% RSLogix 500 project SW2014_AK.RSS, saved by version 12.00.00.00 %
PROJECT "PS8"    % processor: MicroLogix 1400 %

PROGRAM FILES
  LAD 2 "MAIN"  27 rungs  % Calls all system and subsystem routines %
  LAD 3 "CONSTANTS"  51 rungs  % Maintains the system constants %
  LAD 4 "DEFAULTS"  49 rungs  % Manages the system default values %
  LAD 5 "SYS_FAULTS"  43 rungs  % Monitors the system fault conditions %
  LAD 6 "SYSTEM"  50 rungs  % Controls the system %
  LAD 7 "PROCESSING"  33 rungs  % Runs the processing control %
  LAD 8 "MANUAL_CTL"  14 rungs  % Runs the manual valve control %
  LAD 10 "PURIFY"  36 rungs  % Operates the purify control %
  LAD 11 "REGEN"  79 rungs  % Operates the regen control %
  LAD 12 "REGEN_FLT"  47 rungs  % regen alarms and warnings %
  LAD 17 "BYPASS"  4 rungs  % Controls the bypass %
  LAD 18 "MIX PANEL"  9 rungs
  LAD 20 "ADS_A"  45 rungs  % Controls the Adsorber A %
  LAD 21 "ADS_A_FLT"  17 rungs  % Controls the Adsorber A faults %
  LAD 22 "ADS_B"  45 rungs  % Controld Adsorber B %
  LAD 23 "ADS_B_FLT"  17 rungs  % Controls the Adsorber B faults %
  LAD 24 "PREHEATER"  10 rungs
  LAD 25 "PH_FLT"  19 rungs
  LAD 26 "ADS_C"  45 rungs
  LAD 27 "ADS_C_FLT"  17 rungs
  LAD 28 "ADS_D"  45 rungs
  LAD 29 "ADS_D_FLT"  17 rungs
  LAD 49 "MODBUS"  38 rungs
  LAD 50 "PLC_FAULT"  2 rungs
  LAD 51 "REVERSE"  9 rungs

DATA FILES
  O0 OUTPUT  25 elements
  I1 INPUT  25 elements
  S2 STATUS  66 elements
  B3 BINARY  4 elements
  T4 TIMER  142 elements
  C5 COUNTER  22 elements
  R6 CONTROL  2 elements
  N7 SYSTEM CFG  140 elements  % Maintains the values that characterize the system %
  F8 FLOAT  3 elements
  N9 CONSTANTS  86 elements  % The collection of system and subsystem constants %
  N10 SYSTEM  30 elements  % Contain the values for system control %
  N11 PROCESS  10 elements  % Contains the values for the processing machine %
  N12 PURIFY  25 elements  % Contains the values required for purify %
  N13 REGEN  31 elements  % Contains the values required for regen %
  N14 BYPASS  2 elements
  N15 MANUAL CTL  6 elements  % Contains the data for the manual valve control %
  N16 ADSORBER_A  22 elements  % Contains the values for Adsorber A %
  N17 ADSORBER_B  22 elements  % Contains the values required for Adsorber B %
  N18 ADSORBER_C  22 elements
  N19 ADSORBER_D  22 elements
  N20 MIX PANEL  3 elements
  N21 NOMEMBCKUP  4 elements
  T23 MB_HRTBT  3 elements
  PD25 PID HEATER  6 elements
  B30 SYSTEM CFG  7 elements
  B31 SYSTEM  18 elements
  B32 PROCESS  1 elements
  B33 PURIFY  1 elements
  B34 REGEN  5 elements
  B35 MANUAL CTL  6 elements
  B38 HEATERS  1 elements
  L51 TOTAL_FLOW  2 elements
  L52 SERIAL  1 elements
  B54   1 elements
  N64 MODBUS  126 elements
  MG68 TRANSFER  1 elements
  B69 REVERSE  3 elements
  RIX80 MSG_SETUP  1 elements
  N200 STATUS SYS  1 elements
  L201 STATUS PUR  1 elements
  L203 STATUS ADS  4 elements
  F206 FLOAT_PRC  3 elements
  N207 STATUS_PRC  5 elements
  N210 BUZZER  3 elements

LADDER 2 "MAIN"    % Calls all system and subsystem routines %
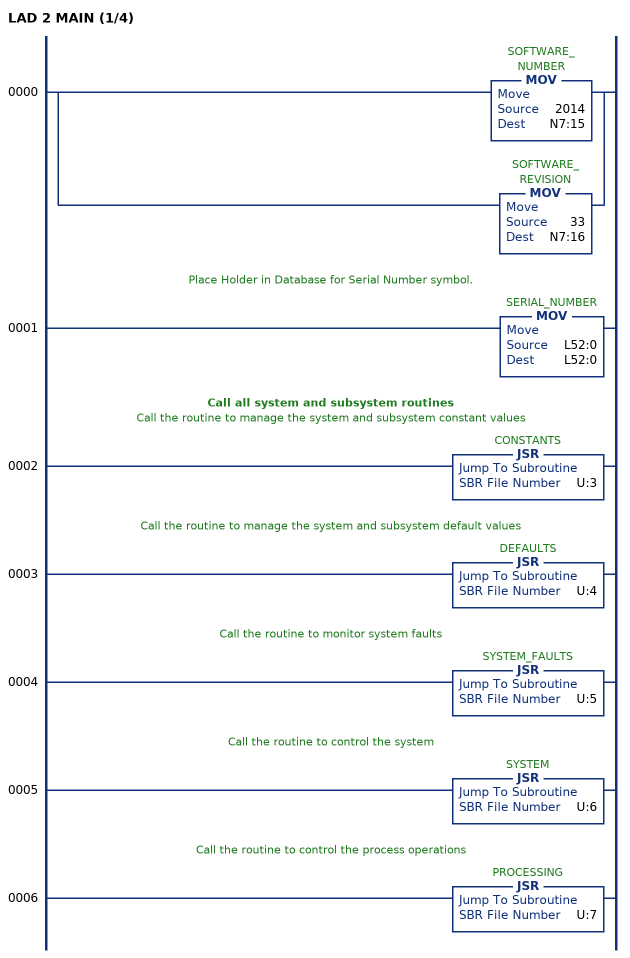
% Rung: 0 %
SOR BST MOV 2014 N7:15 NXB MOV 33 N7:16 BND EOR
%   N7:15  SOFTWARE_NUMBER %
%   N7:16  SOFTWARE_REVISION %
% Rung: 1 %
% Place Holder in Database for Serial Number symbol. %
SOR MOV L52:0 L52:0 EOR
%   L52:0  SERIAL_NUMBER %
% Rung: 2 %
% TITLE: Call all system and subsystem routines %
% Call the routine to manage the system and subsystem constant values %
SOR JSR U:3 EOR
%   U:3  CONSTANTS %
% Rung: 3 %
% Call the routine to manage the system and subsystem default values %
SOR JSR U:4 EOR
%   U:4  DEFAULTS %
% Rung: 4 %
% Call the routine to monitor system faults %
SOR JSR U:5 EOR
%   U:5  SYSTEM_FAULTS %
% Rung: 5 %
% Call the routine to control the system %
SOR JSR U:6 EOR
%   U:6  SYSTEM %
% Rung: 6 %
% Call the routine to control the process operations %
SOR JSR U:7 EOR
%   U:7  PROCESSING %

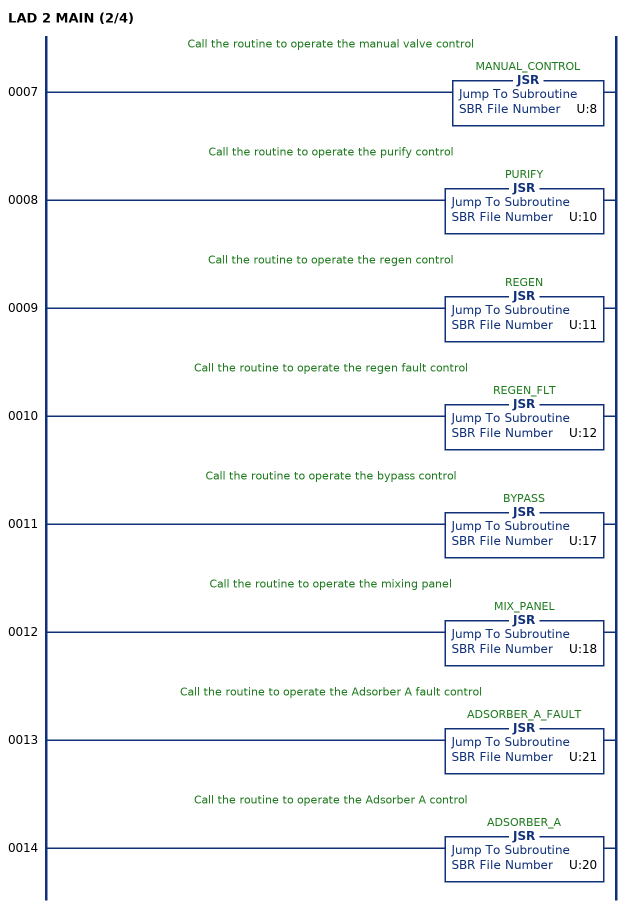
% Rung: 7 %
% Call the routine to operate the manual valve control %
SOR JSR U:8 EOR
%   U:8  MANUAL_CONTROL %
% Rung: 8 %
% Call the routine to operate the purify control %
SOR JSR U:10 EOR
%   U:10  PURIFY %
% Rung: 9 %
% Call the routine to operate the regen control %
SOR JSR U:11 EOR
%   U:11  REGEN %
% Rung: 10 %
% Call the routine to operate the regen fault control %
SOR JSR U:12 EOR
%   U:12  REGEN_FLT %
% Rung: 11 %
% Call the routine to operate the bypass control %
SOR JSR U:17 EOR
%   U:17  BYPASS %
% Rung: 12 %
% Call the routine to operate the mixing panel %
SOR JSR U:18 EOR
%   U:18  MIX_PANEL %
% Rung: 13 %
% Call the routine to operate the Adsorber A fault control %
SOR JSR U:21 EOR
%   U:21  ADSORBER_A_FAULT %
% Rung: 14 %
% Call the routine to operate the Adsorber A control %
SOR JSR U:20 EOR
%   U:20  ADSORBER_A %

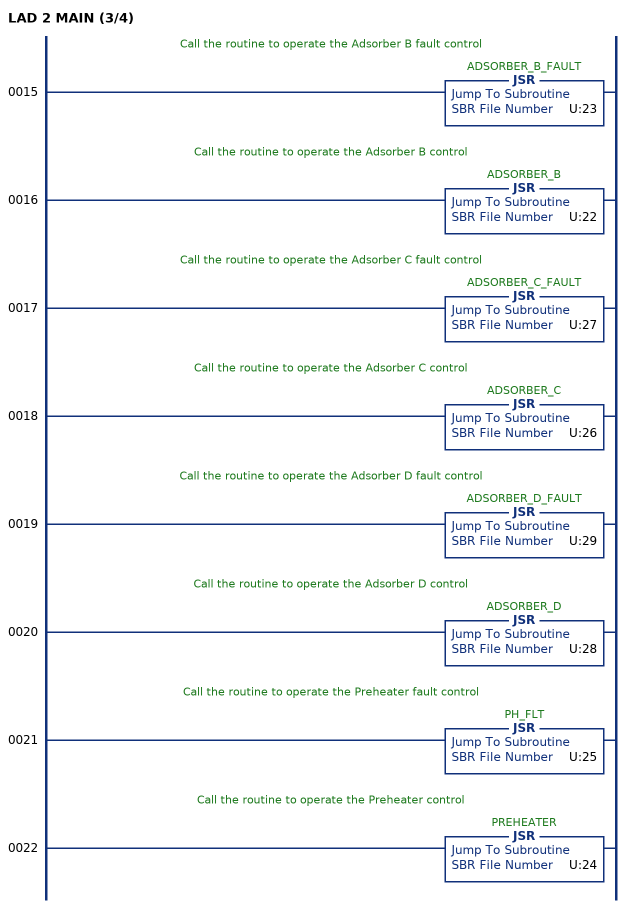
% Rung: 15 %
% Call the routine to operate the Adsorber B fault control %
SOR JSR U:23 EOR
%   U:23  ADSORBER_B_FAULT %
% Rung: 16 %
% Call the routine to operate the Adsorber B control %
SOR JSR U:22 EOR
%   U:22  ADSORBER_B %
% Rung: 17 %
% Call the routine to operate the Adsorber C fault control %
SOR JSR U:27 EOR
%   U:27  ADSORBER_C_FAULT %
% Rung: 18 %
% Call the routine to operate the Adsorber C control %
SOR JSR U:26 EOR
%   U:26  ADSORBER_C %
% Rung: 19 %
% Call the routine to operate the Adsorber D fault control %
SOR JSR U:29 EOR
%   U:29  ADSORBER_D_FAULT %
% Rung: 20 %
% Call the routine to operate the Adsorber D control %
SOR JSR U:28 EOR
%   U:28  ADSORBER_D %
% Rung: 21 %
% Call the routine to operate the Preheater fault control %
SOR JSR U:25 EOR
%   U:25  PH_FLT %
% Rung: 22 %
% Call the routine to operate the Preheater control %
SOR JSR U:24 EOR
%   U:24  PREHEATER %

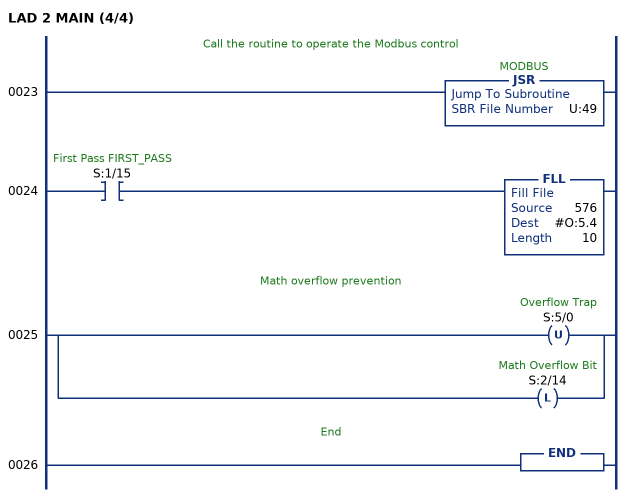
% Rung: 23 %
% Call the routine to operate the Modbus control %
SOR JSR U:49 EOR
%   U:49  MODBUS %
% Rung: 24 %
SOR XIC S:1/15 FLL 576 #O:5.4 10 EOR
%   S:1/15  FIRST_PASS  "First Pass" %
% Rung: 25 %
% Math overflow prevention %
SOR BST OTU S:5/0 NXB OTL S:2/14 BND EOR
%   S:5/0  "Overflow Trap" %
%   S:2/14  "Math Overflow Bit" %
% Rung: 26 %
% End %
SOR END EOR

LADDER 3 "CONSTANTS"    % Maintains the system constants %
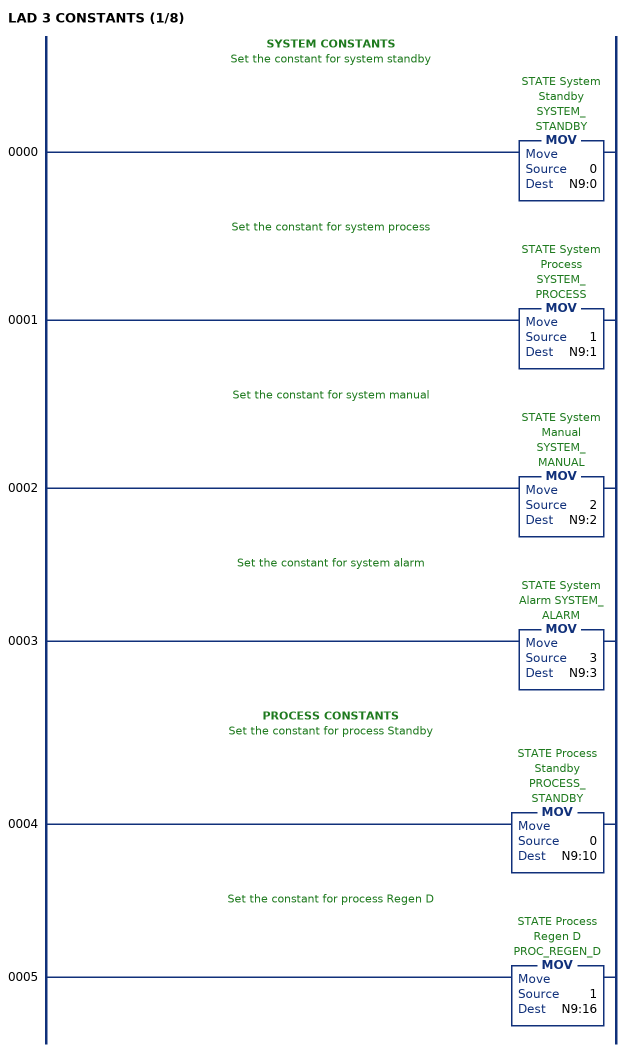
% Rung: 0 %
% TITLE: SYSTEM CONSTANTS %
% Set the constant for system standby %
SOR MOV 0 N9:0 EOR
%   N9:0  SYSTEM_STANDBY  "STATE System Standby" %
% Rung: 1 %
% Set the constant for system process %
SOR MOV 1 N9:1 EOR
%   N9:1  SYSTEM_PROCESS  "STATE System Process" %
% Rung: 2 %
% Set the constant for system manual %
SOR MOV 2 N9:2 EOR
%   N9:2  SYSTEM_MANUAL  "STATE System Manual" %
% Rung: 3 %
% Set the constant for system alarm %
SOR MOV 3 N9:3 EOR
%   N9:3  SYSTEM_ALARM  "STATE System Alarm" %
% Rung: 4 %
% TITLE: PROCESS CONSTANTS %
% Set the constant for process Standby %
SOR MOV 0 N9:10 EOR
%   N9:10  PROCESS_STANDBY  "STATE Process Standby" %
% Rung: 5 %
% Set the constant for process Regen D %
SOR MOV 1 N9:16 EOR
%   N9:16  PROC_REGEN_D  "STATE Process Regen D" %

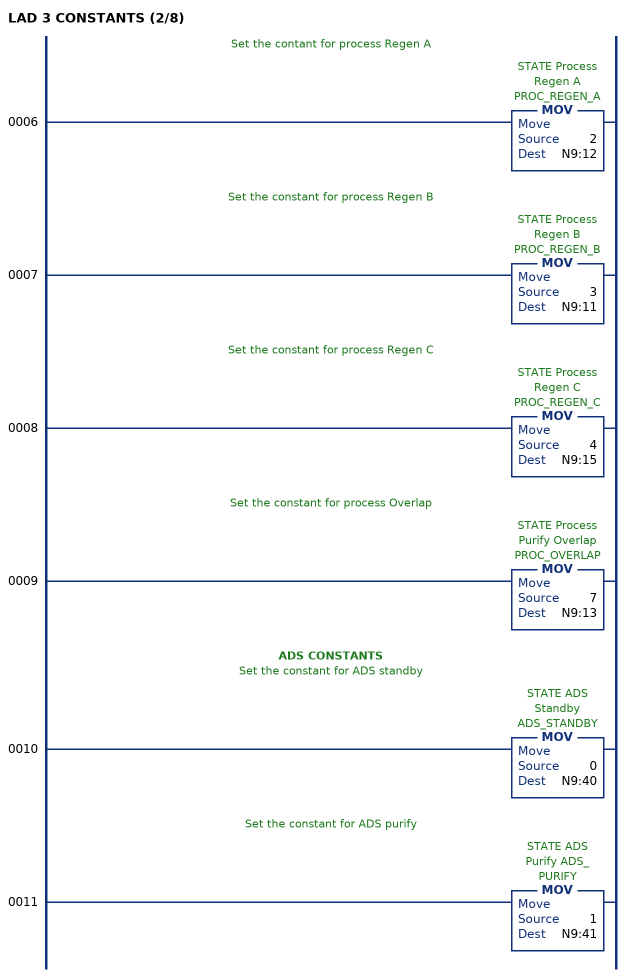
% Rung: 6 %
% Set the contant for process Regen A %
SOR MOV 2 N9:12 EOR
%   N9:12  PROC_REGEN_A  "STATE Process Regen A" %
% Rung: 7 %
% Set the constant for process Regen B %
SOR MOV 3 N9:11 EOR
%   N9:11  PROC_REGEN_B  "STATE Process Regen B" %
% Rung: 8 %
% Set the constant for process Regen C %
SOR MOV 4 N9:15 EOR
%   N9:15  PROC_REGEN_C  "STATE Process Regen C" %
% Rung: 9 %
% Set the constant for process Overlap %
SOR MOV 7 N9:13 EOR
%   N9:13  PROC_OVERLAP  "STATE Process Purify Overlap" %
% Rung: 10 %
% TITLE: ADS CONSTANTS %
% Set the constant for ADS standby %
SOR MOV 0 N9:40 EOR
%   N9:40  ADS_STANDBY  "STATE ADS Standby" %
% Rung: 11 %
% Set the constant for ADS purify %
SOR MOV 1 N9:41 EOR
%   N9:41  ADS_PURIFY  "STATE ADS Purify" %

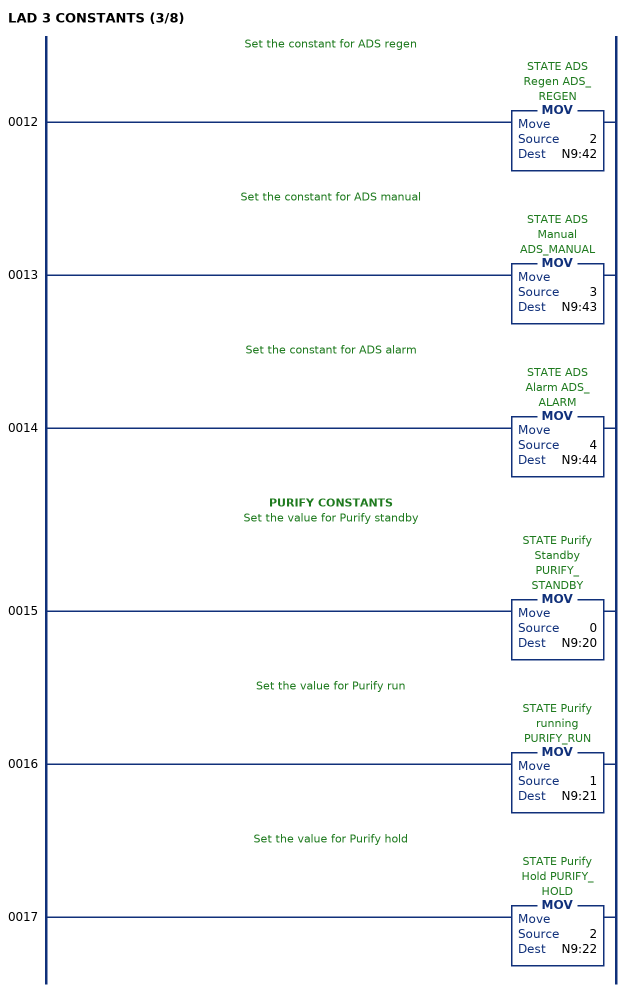
% Rung: 12 %
% Set the constant for ADS regen %
SOR MOV 2 N9:42 EOR
%   N9:42  ADS_REGEN  "STATE ADS Regen" %
% Rung: 13 %
% Set the constant for ADS manual %
SOR MOV 3 N9:43 EOR
%   N9:43  ADS_MANUAL  "STATE ADS Manual" %
% Rung: 14 %
% Set the constant for ADS alarm %
SOR MOV 4 N9:44 EOR
%   N9:44  ADS_ALARM  "STATE ADS Alarm" %
% Rung: 15 %
% TITLE: PURIFY CONSTANTS %
% Set the value for Purify standby %
SOR MOV 0 N9:20 EOR
%   N9:20  PURIFY_STANDBY  "STATE Purify Standby" %
% Rung: 16 %
% Set the value for Purify run %
SOR MOV 1 N9:21 EOR
%   N9:21  PURIFY_RUN  "STATE Purify running" %
% Rung: 17 %
% Set the value for Purify hold %
SOR MOV 2 N9:22 EOR
%   N9:22  PURIFY_HOLD  "STATE Purify Hold" %

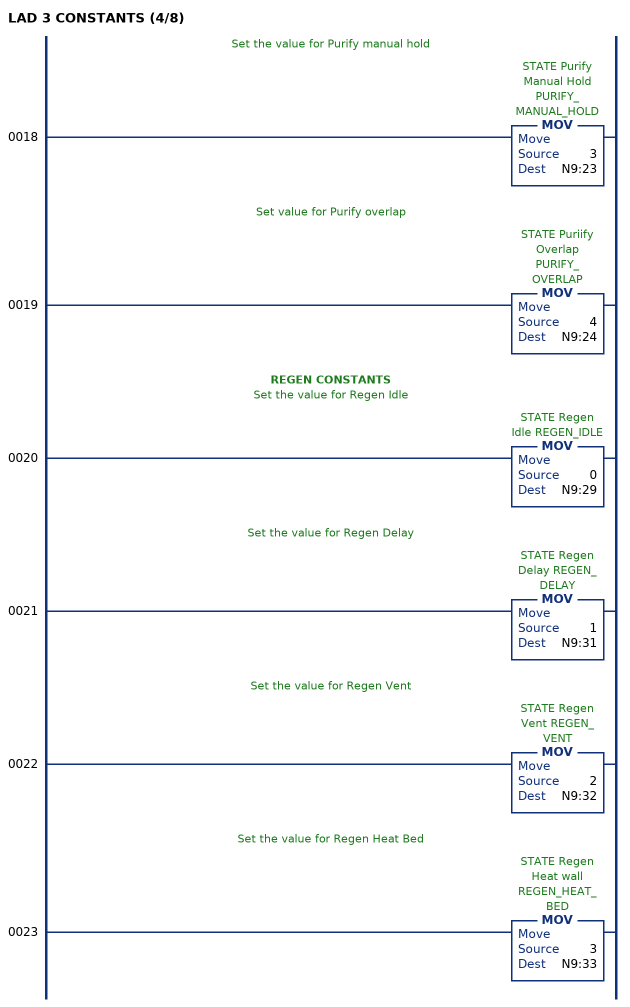
% Rung: 18 %
% Set the value for Purify manual hold %
SOR MOV 3 N9:23 EOR
%   N9:23  PURIFY_MANUAL_HOLD  "STATE Purify Manual Hold" %
% Rung: 19 %
% Set value for Purify overlap %
SOR MOV 4 N9:24 EOR
%   N9:24  PURIFY_OVERLAP  "STATE Puriify Overlap" %
% Rung: 20 %
% TITLE: REGEN CONSTANTS %
% Set the value for Regen Idle %
SOR MOV 0 N9:29 EOR
%   N9:29  REGEN_IDLE  "STATE Regen Idle" %
% Rung: 21 %
% Set the value for Regen Delay %
SOR MOV 1 N9:31 EOR
%   N9:31  REGEN_DELAY  "STATE Regen Delay" %
% Rung: 22 %
% Set the value for Regen Vent %
SOR MOV 2 N9:32 EOR
%   N9:32  REGEN_VENT  "STATE Regen Vent" %
% Rung: 23 %
% Set the value for Regen Heat Bed %
SOR MOV 3 N9:33 EOR
%   N9:33  REGEN_HEAT_BED  "STATE Regen Heat wall" %

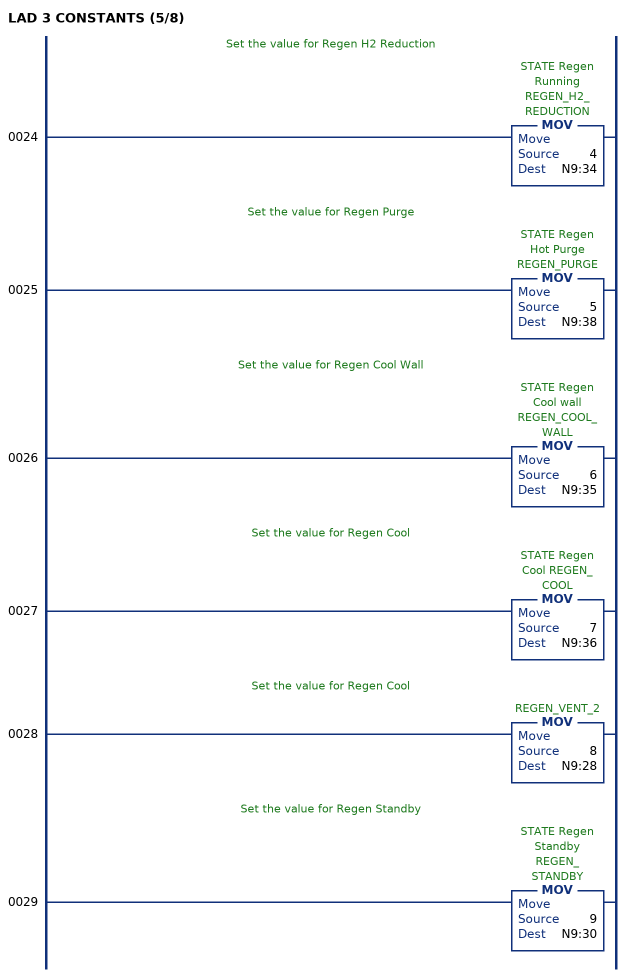
% Rung: 24 %
% Set the value for Regen H2 Reduction %
SOR MOV 4 N9:34 EOR
%   N9:34  REGEN_H2_REDUCTION  "STATE Regen Running" %
% Rung: 25 %
% Set the value for Regen Purge %
SOR MOV 5 N9:38 EOR
%   N9:38  REGEN_PURGE  "STATE Regen Hot Purge" %
% Rung: 26 %
% Set the value for Regen Cool Wall %
SOR MOV 6 N9:35 EOR
%   N9:35  REGEN_COOL_WALL  "STATE Regen Cool wall" %
% Rung: 27 %
% Set the value for Regen Cool %
SOR MOV 7 N9:36 EOR
%   N9:36  REGEN_COOL  "STATE Regen Cool" %
% Rung: 28 %
% Set the value for Regen Cool %
SOR MOV 8 N9:28 EOR
%   N9:28  REGEN_VENT_2 %
% Rung: 29 %
% Set the value for Regen Standby %
SOR MOV 9 N9:30 EOR
%   N9:30  REGEN_STANDBY  "STATE Regen Standby" %

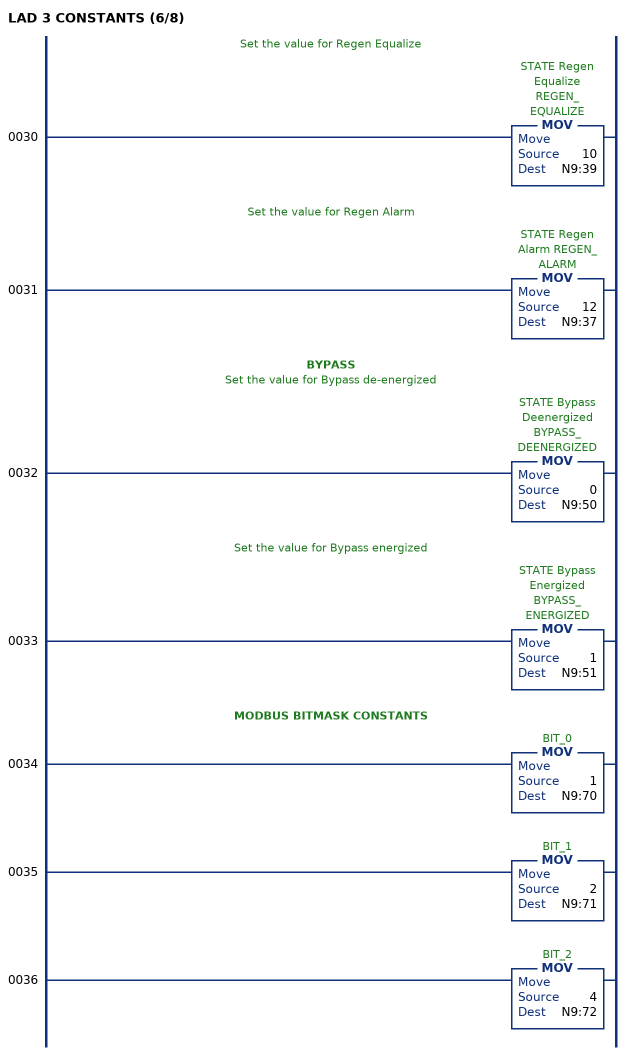
% Rung: 30 %
% Set the value for Regen Equalize %
SOR MOV 10 N9:39 EOR
%   N9:39  REGEN_EQUALIZE  "STATE Regen Equalize" %
% Rung: 31 %
% Set the value for Regen Alarm %
SOR MOV 12 N9:37 EOR
%   N9:37  REGEN_ALARM  "STATE Regen Alarm" %
% Rung: 32 %
% TITLE: BYPASS %
% Set the value for Bypass de-energized %
SOR MOV 0 N9:50 EOR
%   N9:50  BYPASS_DEENERGIZED  "STATE Bypass Deenergized" %
% Rung: 33 %
% Set the value for Bypass energized %
SOR MOV 1 N9:51 EOR
%   N9:51  BYPASS_ENERGIZED  "STATE Bypass Energized" %
% Rung: 34 %
% TITLE: MODBUS BITMASK CONSTANTS %
SOR MOV 1 N9:70 EOR
%   N9:70  BIT_0 %
% Rung: 35 %
SOR MOV 2 N9:71 EOR
%   N9:71  BIT_1 %
% Rung: 36 %
SOR MOV 4 N9:72 EOR
%   N9:72  BIT_2 %

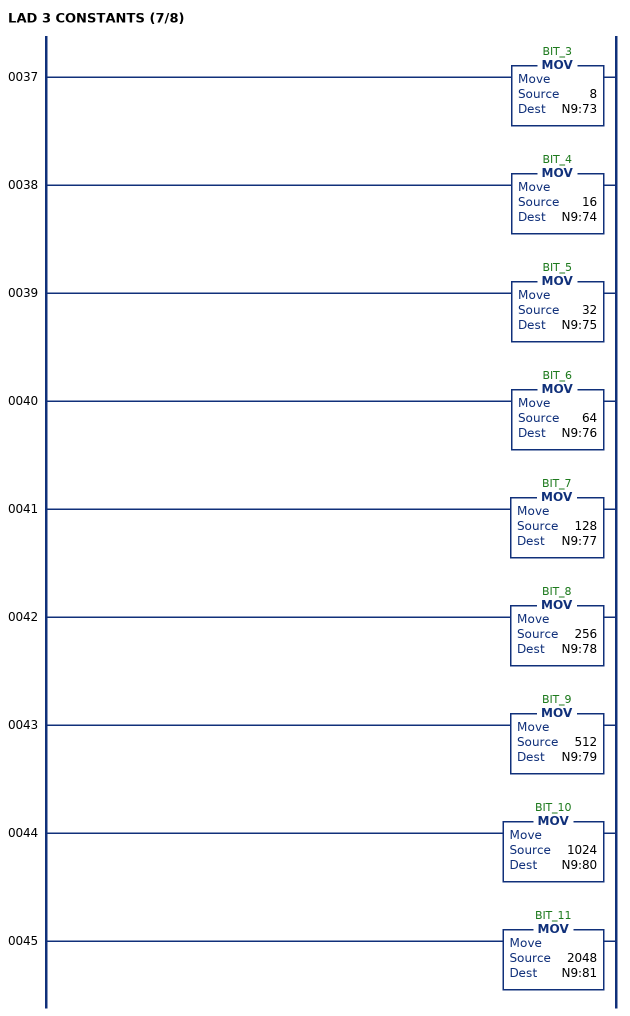
% Rung: 37 %
SOR MOV 8 N9:73 EOR
%   N9:73  BIT_3 %
% Rung: 38 %
SOR MOV 16 N9:74 EOR
%   N9:74  BIT_4 %
% Rung: 39 %
SOR MOV 32 N9:75 EOR
%   N9:75  BIT_5 %
% Rung: 40 %
SOR MOV 64 N9:76 EOR
%   N9:76  BIT_6 %
% Rung: 41 %
SOR MOV 128 N9:77 EOR
%   N9:77  BIT_7 %
% Rung: 42 %
SOR MOV 256 N9:78 EOR
%   N9:78  BIT_8 %
% Rung: 43 %
SOR MOV 512 N9:79 EOR
%   N9:79  BIT_9 %
% Rung: 44 %
SOR MOV 1024 N9:80 EOR
%   N9:80  BIT_10 %
% Rung: 45 %
SOR MOV 2048 N9:81 EOR
%   N9:81  BIT_11 %

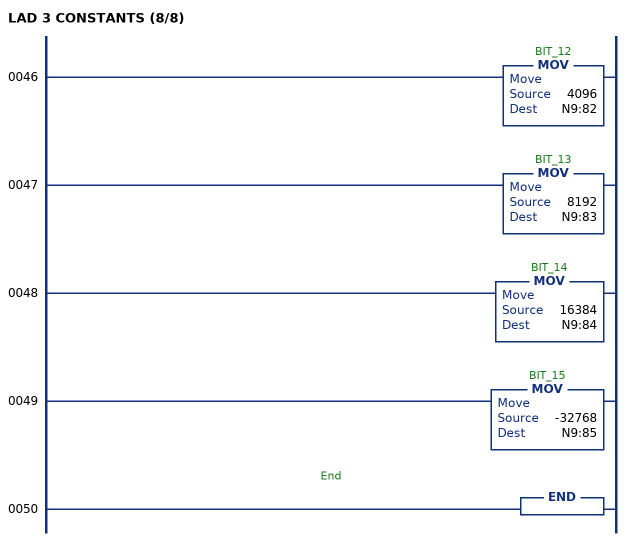
% Rung: 46 %
SOR MOV 4096 N9:82 EOR
%   N9:82  BIT_12 %
% Rung: 47 %
SOR MOV 8192 N9:83 EOR
%   N9:83  BIT_13 %
% Rung: 48 %
SOR MOV 16384 N9:84 EOR
%   N9:84  BIT_14 %
% Rung: 49 %
SOR MOV -32768 N9:85 EOR
%   N9:85  BIT_15 %
% Rung: 50 %
% End %
SOR END EOR

LADDER 4 "DEFAULTS"    % Manages the system default values %
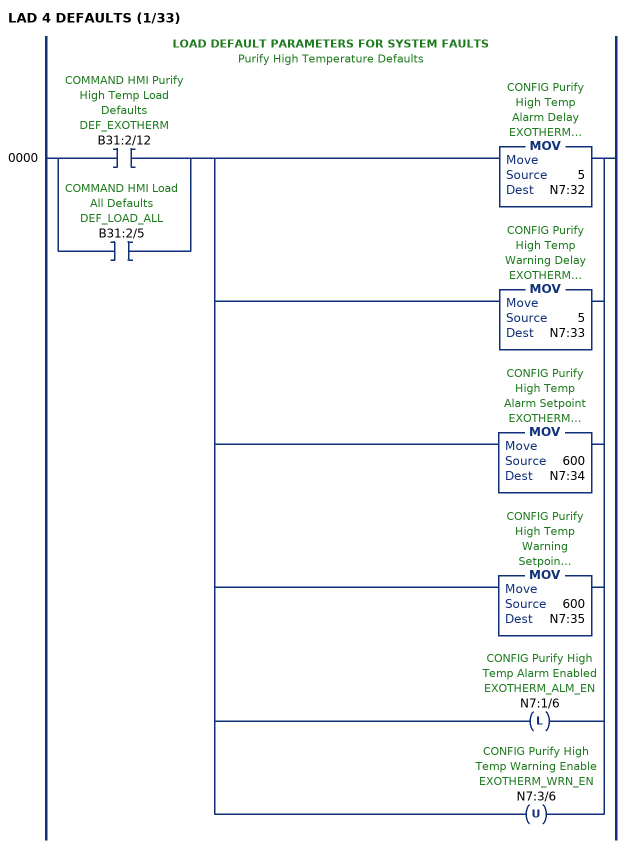
% Rung: 0 %
% TITLE: LOAD DEFAULT PARAMETERS FOR SYSTEM FAULTS %
% Purify High Temperature Defaults %
SOR BST XIC B31:2/12 NXB XIC B31:2/5 BND BST MOV 5 N7:32 NXB MOV 5 N7:33 NXB MOV 600 N7:34 NXB MOV 600 N7:35 NXB OTL N7:1/6 NXB OTU N7:3/6 BND EOR
%   B31:2/12  DEF_EXOTHERM  "COMMAND HMI Purify High Temp Load Defaults" %
%   B31:2/5  DEF_LOAD_ALL  "COMMAND HMI Load All Defaults" %
%   N7:32  EXOTHERM_ALM_DLY  "CONFIG Purify High Temp Alarm Delay" %
%   N7:33  EXOTHERM_WRN_DLY  "CONFIG Purify High Temp Warning Delay" %
%   N7:34  EXOTHERM_ALM_SP  "CONFIG Purify High Temp Alarm Setpoint" %
%   N7:35  EXOTHERM_WRN_SP  "CONFIG Purify High Temp Warning Setpoint" %
%   N7:1/6  EXOTHERM_ALM_EN  "CONFIG Purify High Temp Alarm Enabled" %
%   N7:3/6  EXOTHERM_WRN_EN  "CONFIG Purify High Temp Warning Enable" %

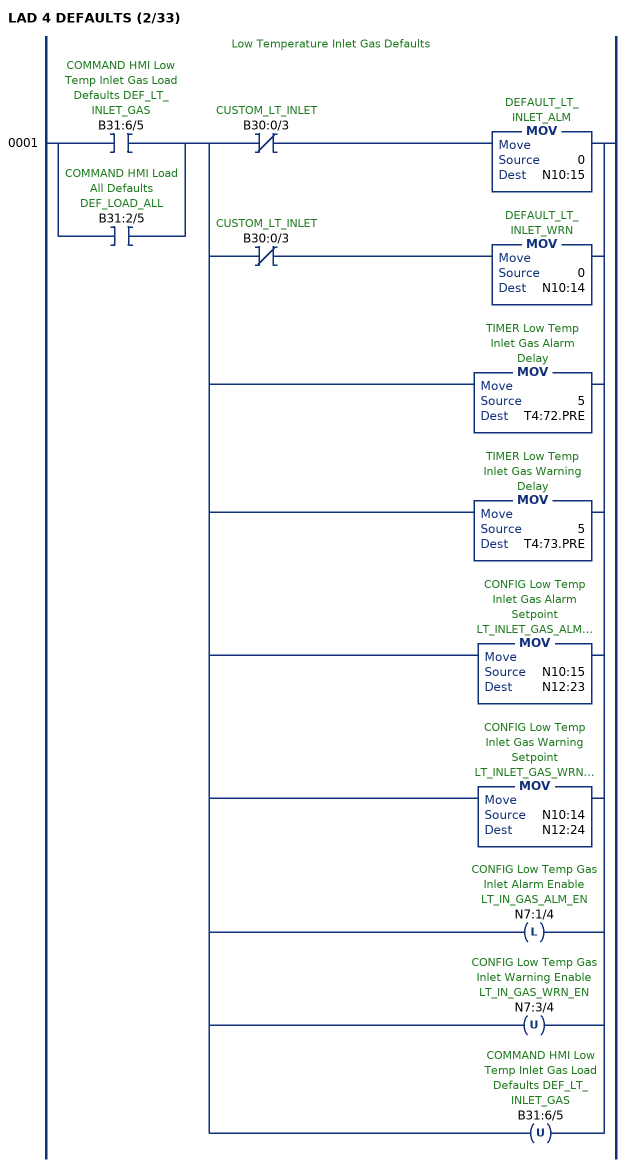
% Rung: 1 %
% Low Temperature Inlet Gas Defaults %
SOR BST XIC B31:6/5 NXB XIC B31:2/5 BND BST XIO B30:0/3 MOV 0 N10:15 NXB XIO B30:0/3 MOV 0 N10:14 NXB MOV 5 T4:72.PRE NXB MOV 5 T4:73.PRE NXB MOV N10:15 N12:23 NXB MOV N10:14 N12:24 NXB OTL N7:1/4 NXB OTU N7:3/4 NXB OTU B31:6/5 BND EOR
%   B31:6/5  DEF_LT_INLET_GAS  "COMMAND HMI Low Temp Inlet Gas Load Defaults" %
%   B31:2/5  DEF_LOAD_ALL  "COMMAND HMI Load All Defaults" %
%   B30:0/3  CUSTOM_LT_INLET %
%   N10:15  DEFAULT_LT_INLET_ALM %
%   N10:14  DEFAULT_LT_INLET_WRN %
%   T4:72.PRE  "TIMER Low Temp Inlet Gas Alarm Delay" %
%   T4:73.PRE  "TIMER Low Temp Inlet Gas Warning Delay" %
%   N12:23  LT_INLET_GAS_ALM_SP  "CONFIG Low Temp Inlet Gas Alarm Setpoint" %
%   N12:24  LT_INLET_GAS_WRN_SP  "CONFIG Low Temp Inlet Gas Warning Setpoint" %
%   N7:1/4  LT_IN_GAS_ALM_EN  "CONFIG Low Temp Gas Inlet Alarm Enable" %
%   N7:3/4  LT_IN_GAS_WRN_EN  "CONFIG Low Temp Gas Inlet Warning Enable" %

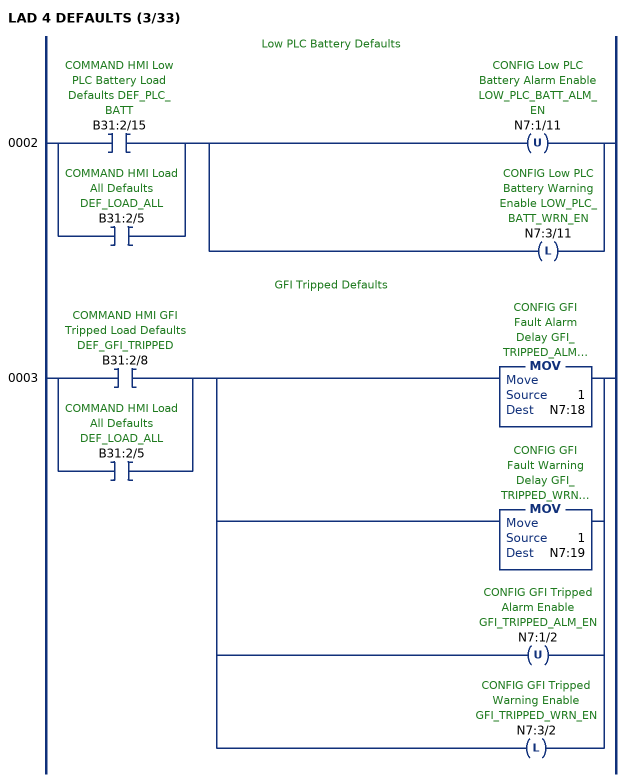
% Rung: 2 %
% Low PLC Battery Defaults %
SOR BST XIC B31:2/15 NXB XIC B31:2/5 BND BST OTU N7:1/11 NXB OTL N7:3/11 BND EOR
%   B31:2/15  DEF_PLC_BATT  "COMMAND HMI Low PLC Battery Load Defaults" %
%   B31:2/5  DEF_LOAD_ALL  "COMMAND HMI Load All Defaults" %
%   N7:1/11  LOW_PLC_BATT_ALM_EN  "CONFIG Low PLC Battery Alarm Enable" %
%   N7:3/11  LOW_PLC_BATT_WRN_EN  "CONFIG Low PLC Battery Warning Enable" %
% Rung: 3 %
% GFI Tripped Defaults %
SOR BST XIC B31:2/8 NXB XIC B31:2/5 BND BST MOV 1 N7:18 NXB MOV 1 N7:19 NXB OTU N7:1/2 NXB OTL N7:3/2 BND EOR
%   B31:2/8  DEF_GFI_TRIPPED  "COMMAND HMI GFI Tripped Load Defaults" %
%   B31:2/5  DEF_LOAD_ALL  "COMMAND HMI Load All Defaults" %
%   N7:18  GFI_TRIPPED_ALM_DLY  "CONFIG GFI Fault Alarm Delay" %
%   N7:19  GFI_TRIPPED_WRN_DLY  "CONFIG GFI Fault Warning Delay" %
%   N7:1/2  GFI_TRIPPED_ALM_EN  "CONFIG GFI Tripped Alarm Enable" %
%   N7:3/2  GFI_TRIPPED_WRN_EN  "CONFIG GFI Tripped Warning Enable" %

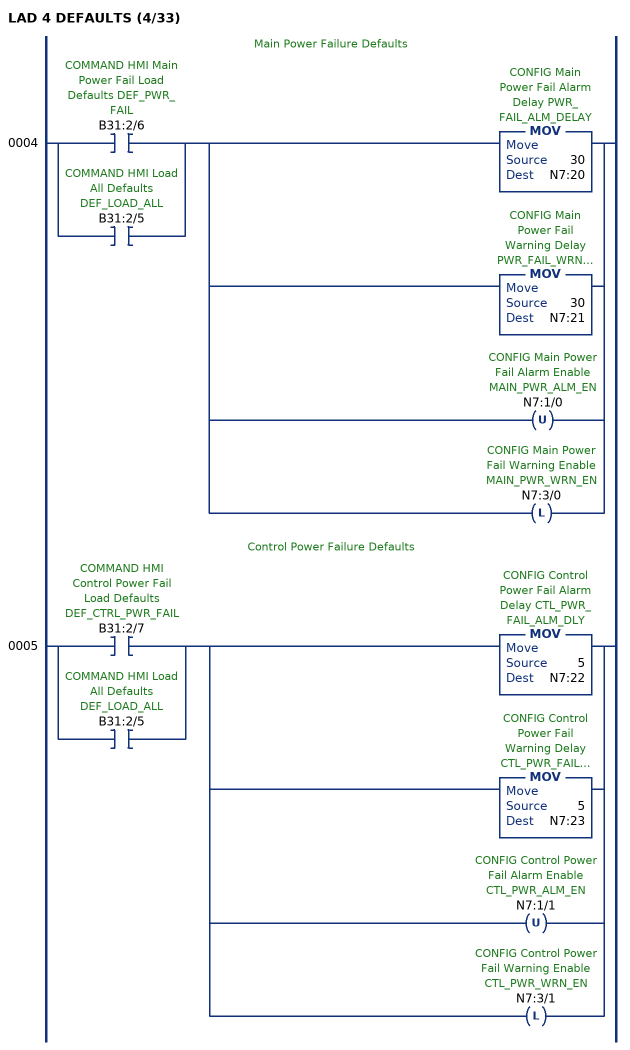
% Rung: 4 %
% Main Power Failure Defaults %
SOR BST XIC B31:2/6 NXB XIC B31:2/5 BND BST MOV 30 N7:20 NXB MOV 30 N7:21 NXB OTU N7:1/0 NXB OTL N7:3/0 BND EOR
%   B31:2/6  DEF_PWR_FAIL  "COMMAND HMI Main Power Fail Load Defaults" %
%   B31:2/5  DEF_LOAD_ALL  "COMMAND HMI Load All Defaults" %
%   N7:20  PWR_FAIL_ALM_DELAY  "CONFIG Main Power Fail Alarm Delay" %
%   N7:21  PWR_FAIL_WRN_DELAY  "CONFIG Main Power Fail Warning Delay" %
%   N7:1/0  MAIN_PWR_ALM_EN  "CONFIG Main Power Fail Alarm Enable" %
%   N7:3/0  MAIN_PWR_WRN_EN  "CONFIG Main Power Fail Warning Enable" %
% Rung: 5 %
% Control Power Failure Defaults %
SOR BST XIC B31:2/7 NXB XIC B31:2/5 BND BST MOV 5 N7:22 NXB MOV 5 N7:23 NXB OTU N7:1/1 NXB OTL N7:3/1 BND EOR
%   B31:2/7  DEF_CTRL_PWR_FAIL  "COMMAND HMI Control Power Fail Load Defaults" %
%   B31:2/5  DEF_LOAD_ALL  "COMMAND HMI Load All Defaults" %
%   N7:22  CTL_PWR_FAIL_ALM_DLY  "CONFIG Control Power Fail Alarm Delay" %
%   N7:23  CTL_PWR_FAIL_WRN_DLY  "CONFIG Control Power Fail Warning Delay" %
%   N7:1/1  CTL_PWR_ALM_EN  "CONFIG Control Power Fail Alarm Enable" %
%   N7:3/1  CTL_PWR_WRN_EN  "CONFIG Control Power Fail Warning Enable" %

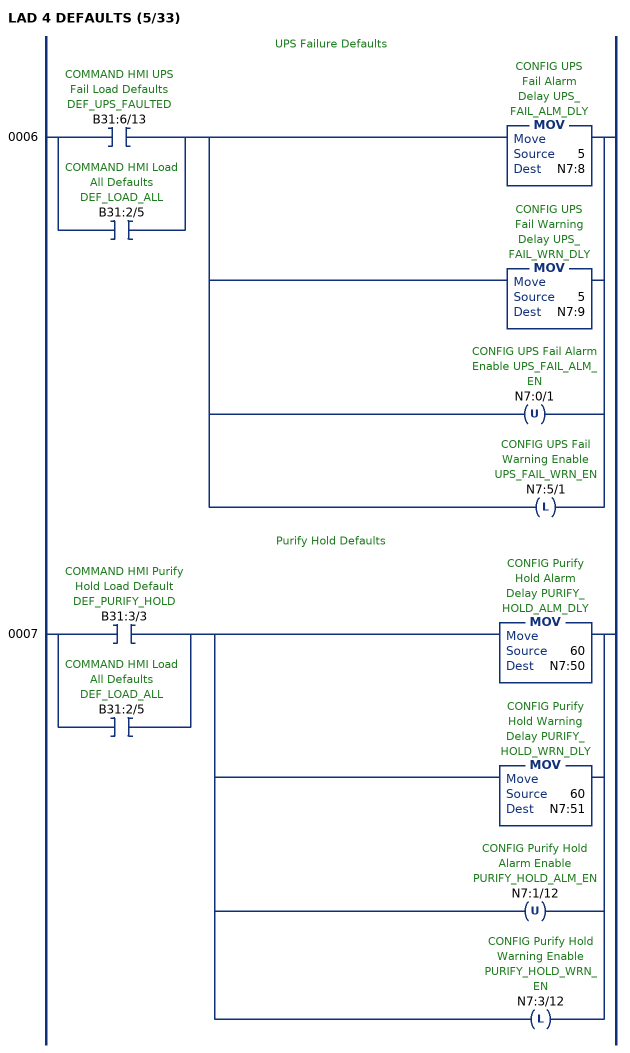
% Rung: 6 %
% UPS Failure Defaults %
SOR BST XIC B31:6/13 NXB XIC B31:2/5 BND BST MOV 5 N7:8 NXB MOV 5 N7:9 NXB OTU N7:0/1 NXB OTL N7:5/1 BND EOR
%   B31:6/13  DEF_UPS_FAULTED  "COMMAND HMI UPS Fail Load Defaults" %
%   B31:2/5  DEF_LOAD_ALL  "COMMAND HMI Load All Defaults" %
%   N7:8  UPS_FAIL_ALM_DLY  "CONFIG UPS Fail Alarm Delay" %
%   N7:9  UPS_FAIL_WRN_DLY  "CONFIG UPS Fail Warning Delay" %
%   N7:0/1  UPS_FAIL_ALM_EN  "CONFIG UPS Fail Alarm Enable" %
%   N7:5/1  UPS_FAIL_WRN_EN  "CONFIG UPS Fail Warning Enable" %
% Rung: 7 %
% Purify Hold Defaults %
SOR BST XIC B31:3/3 NXB XIC B31:2/5 BND BST MOV 60 N7:50 NXB MOV 60 N7:51 NXB OTU N7:1/12 NXB OTL N7:3/12 BND EOR
%   B31:3/3  DEF_PURIFY_HOLD  "COMMAND HMI Purify Hold Load Default" %
%   B31:2/5  DEF_LOAD_ALL  "COMMAND HMI Load All Defaults" %
%   N7:50  PURIFY_HOLD_ALM_DLY  "CONFIG Purify Hold Alarm Delay" %
%   N7:51  PURIFY_HOLD_WRN_DLY  "CONFIG Purify Hold Warning Delay" %
%   N7:1/12  PURIFY_HOLD_ALM_EN  "CONFIG Purify Hold Alarm Enable" %
%   N7:3/12  PURIFY_HOLD_WRN_EN  "CONFIG Purify Hold Warning Enable" %

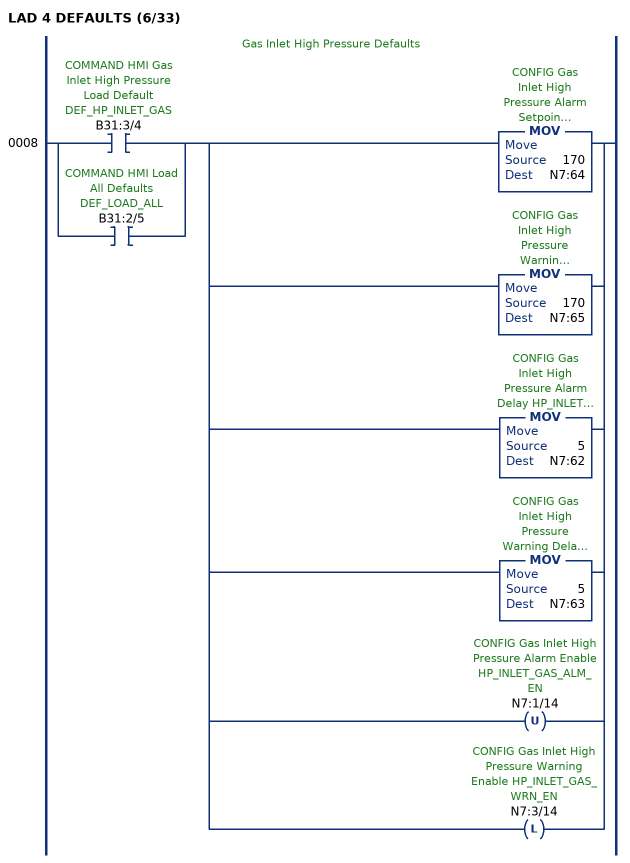
% Rung: 8 %
% Gas Inlet High Pressure Defaults %
SOR BST XIC B31:3/4 NXB XIC B31:2/5 BND BST MOV 170 N7:64 NXB MOV 170 N7:65 NXB MOV 5 N7:62 NXB MOV 5 N7:63 NXB OTU N7:1/14 NXB OTL N7:3/14 BND EOR
%   B31:3/4  DEF_HP_INLET_GAS  "COMMAND HMI Gas Inlet High Pressure Load Default" %
%   B31:2/5  DEF_LOAD_ALL  "COMMAND HMI Load All Defaults" %
%   N7:64  HP_INLET_GAS_ALM_SP  "CONFIG Gas Inlet High Pressure Alarm Setpoint" %
%   N7:65  HP_INLET_GAS_WRN_SP  "CONFIG Gas Inlet High Pressure Warning Setpoint" %
%   N7:62  HP_INLET_GAS_ALM_DLY  "CONFIG Gas Inlet High Pressure Alarm Delay" %
%   N7:63  HP_INLET_GAS_WRN_DLY  "CONFIG Gas Inlet High Pressure Warning Delay" %
%   N7:1/14  HP_INLET_GAS_ALM_EN  "CONFIG Gas Inlet High Pressure Alarm Enable" %
%   N7:3/14  HP_INLET_GAS_WRN_EN  "CONFIG Gas Inlet High Pressure Warning Enable" %

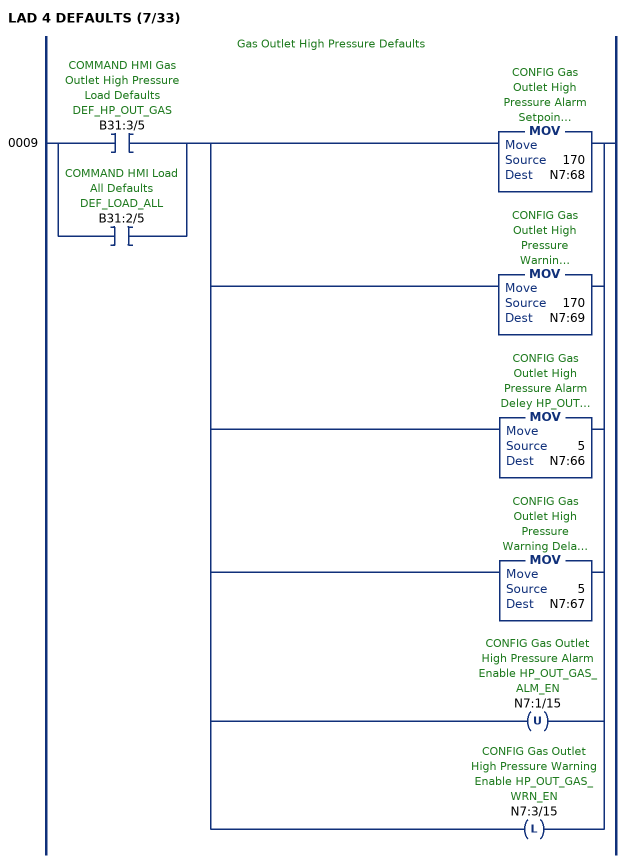
% Rung: 9 %
% Gas Outlet High Pressure Defaults %
SOR BST XIC B31:3/5 NXB XIC B31:2/5 BND BST MOV 170 N7:68 NXB MOV 170 N7:69 NXB MOV 5 N7:66 NXB MOV 5 N7:67 NXB OTU N7:1/15 NXB OTL N7:3/15 BND EOR
%   B31:3/5  DEF_HP_OUT_GAS  "COMMAND HMI Gas Outlet High Pressure Load Defaults" %
%   B31:2/5  DEF_LOAD_ALL  "COMMAND HMI Load All Defaults" %
%   N7:68  HP_OUT_GAS_ALM_SP  "CONFIG Gas Outlet High Pressure Alarm Setpoint" %
%   N7:69  HP_OUT_GAS_WRN_SP  "CONFIG Gas Outlet High Pressure Warning Setpoint" %
%   N7:66  HP_OUT_GAS_ALM_DLY  "CONFIG Gas Outlet High Pressure Alarm Deley" %
%   N7:67  HP_OUT_GAS_WRN_DLY  "CONFIG Gas Outlet High Pressure Warning Delay" %
%   N7:1/15  HP_OUT_GAS_ALM_EN  "CONFIG Gas Outlet High Pressure Alarm Enable" %
%   N7:3/15  HP_OUT_GAS_WRN_EN  "CONFIG Gas Outlet High Pressure Warning Enable" %

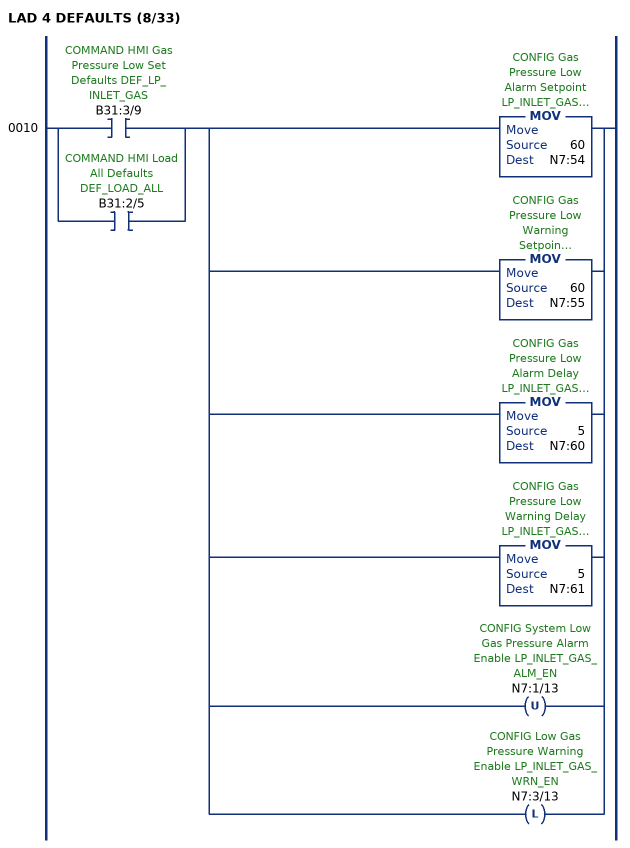
% Rung: 10 %
SOR BST XIC B31:3/9 NXB XIC B31:2/5 BND BST MOV 60 N7:54 NXB MOV 60 N7:55 NXB MOV 5 N7:60 NXB MOV 5 N7:61 NXB OTU N7:1/13 NXB OTL N7:3/13 BND EOR
%   B31:3/9  DEF_LP_INLET_GAS  "COMMAND HMI Gas Pressure Low Set Defaults" %
%   B31:2/5  DEF_LOAD_ALL  "COMMAND HMI Load All Defaults" %
%   N7:54  LP_INLET_GAS_ALM_SP  "CONFIG Gas Pressure Low Alarm Setpoint" %
%   N7:55  LP_INLET_GAS_WRN_SP  "CONFIG Gas Pressure Low Warning Setpoint" %
%   N7:60  LP_INLET_GAS_ALM_DLY  "CONFIG Gas Pressure Low Alarm Delay" %
%   N7:61  LP_INLET_GAS_WRN_DLY  "CONFIG Gas Pressure Low Warning Delay" %
%   N7:1/13  LP_INLET_GAS_ALM_EN  "CONFIG System Low Gas Pressure Alarm Enable" %
%   N7:3/13  LP_INLET_GAS_WRN_EN  "CONFIG Low Gas Pressure Warning Enable" %

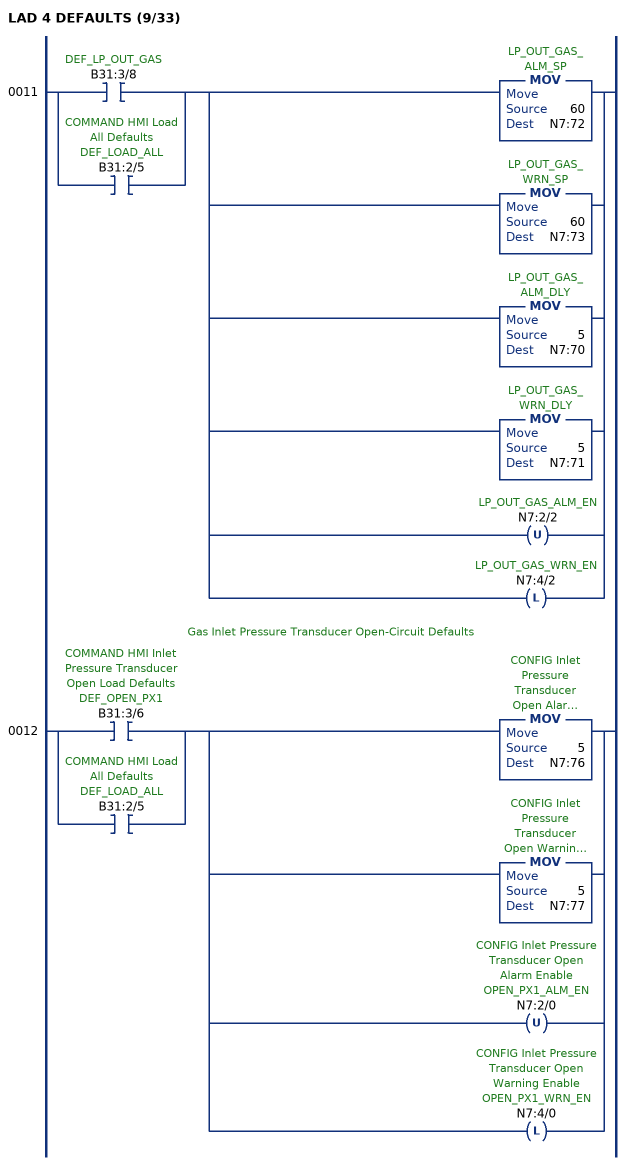
% Rung: 11 %
SOR BST XIC B31:3/8 NXB XIC B31:2/5 BND BST MOV 60 N7:72 NXB MOV 60 N7:73 NXB MOV 5 N7:70 NXB MOV 5 N7:71 NXB OTU N7:2/2 NXB OTL N7:4/2 BND EOR
%   B31:3/8  DEF_LP_OUT_GAS %
%   B31:2/5  DEF_LOAD_ALL  "COMMAND HMI Load All Defaults" %
%   N7:72  LP_OUT_GAS_ALM_SP %
%   N7:73  LP_OUT_GAS_WRN_SP %
%   N7:70  LP_OUT_GAS_ALM_DLY %
%   N7:71  LP_OUT_GAS_WRN_DLY %
%   N7:2/2  LP_OUT_GAS_ALM_EN %
%   N7:4/2  LP_OUT_GAS_WRN_EN %
% Rung: 12 %
% Gas Inlet Pressure Transducer Open-Circuit Defaults %
SOR BST XIC B31:3/6 NXB XIC B31:2/5 BND BST MOV 5 N7:76 NXB MOV 5 N7:77 NXB OTU N7:2/0 NXB OTL N7:4/0 BND EOR
%   B31:3/6  DEF_OPEN_PX1  "COMMAND HMI Inlet Pressure Transducer Open Load Defaults" %
%   B31:2/5  DEF_LOAD_ALL  "COMMAND HMI Load All Defaults" %
%   N7:76  OPEN_PX1_ALM_DLY  "CONFIG Inlet Pressure Transducer Open Alarm Delay" %
%   N7:77  OPEN_PX1_WRN_DLY  "CONFIG Inlet Pressure Transducer Open Warning Delay" %
%   N7:2/0  OPEN_PX1_ALM_EN  "CONFIG Inlet Pressure Transducer Open Alarm Enable" %
%   N7:4/0  OPEN_PX1_WRN_EN  "CONFIG Inlet Pressure Transducer Open Warning Enable" %

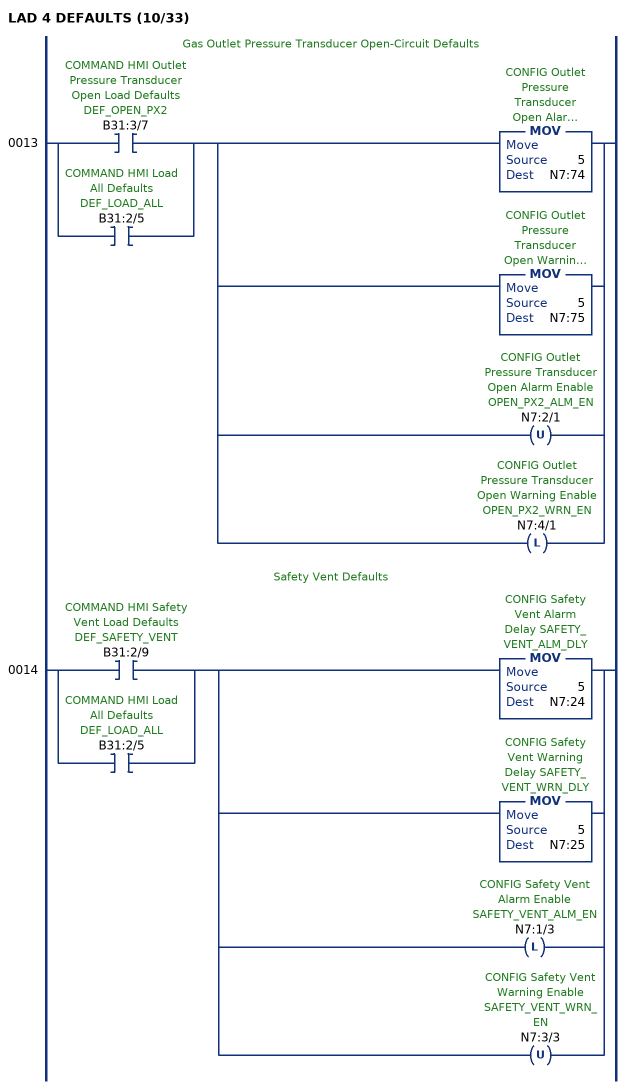
% Rung: 13 %
% Gas Outlet Pressure Transducer Open-Circuit Defaults %
SOR BST XIC B31:3/7 NXB XIC B31:2/5 BND BST MOV 5 N7:74 NXB MOV 5 N7:75 NXB OTU N7:2/1 NXB OTL N7:4/1 BND EOR
%   B31:3/7  DEF_OPEN_PX2  "COMMAND HMI Outlet Pressure Transducer Open Load Defaults" %
%   B31:2/5  DEF_LOAD_ALL  "COMMAND HMI Load All Defaults" %
%   N7:74  OPEN_PX2_ALM_DLY  "CONFIG Outlet Pressure Transducer Open Alarm Delay" %
%   N7:75  OPEN_PX2_WRN_DLY  "CONFIG Outlet Pressure Transducer Open Warning Delay" %
%   N7:2/1  OPEN_PX2_ALM_EN  "CONFIG Outlet Pressure Transducer Open Alarm Enable" %
%   N7:4/1  OPEN_PX2_WRN_EN  "CONFIG Outlet Pressure Transducer Open Warning Enable" %
% Rung: 14 %
% Safety Vent Defaults %
SOR BST XIC B31:2/9 NXB XIC B31:2/5 BND BST MOV 5 N7:24 NXB MOV 5 N7:25 NXB OTL N7:1/3 NXB OTU N7:3/3 BND EOR
%   B31:2/9  DEF_SAFETY_VENT  "COMMAND HMI Safety Vent Load Defaults" %
%   B31:2/5  DEF_LOAD_ALL  "COMMAND HMI Load All Defaults" %
%   N7:24  SAFETY_VENT_ALM_DLY  "CONFIG Safety Vent Alarm Delay" %
%   N7:25  SAFETY_VENT_WRN_DLY  "CONFIG Safety Vent Warning Delay" %
%   N7:1/3  SAFETY_VENT_ALM_EN  "CONFIG Safety Vent Alarm Enable" %
%   N7:3/3  SAFETY_VENT_WRN_EN  "CONFIG Safety Vent Warning Enable" %

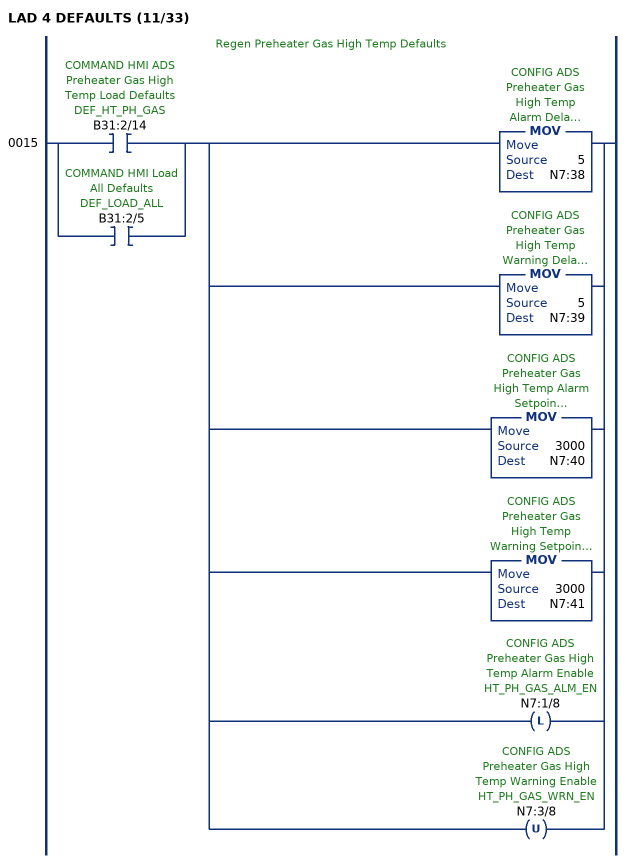
% Rung: 15 %
% Regen Preheater Gas High Temp Defaults %
SOR BST XIC B31:2/14 NXB XIC B31:2/5 BND BST MOV 5 N7:38 NXB MOV 5 N7:39 NXB MOV 3000 N7:40 NXB MOV 3000 N7:41 NXB OTL N7:1/8 NXB OTU N7:3/8 BND EOR
%   B31:2/14  DEF_HT_PH_GAS  "COMMAND HMI ADS Preheater Gas High Temp Load Defaults" %
%   B31:2/5  DEF_LOAD_ALL  "COMMAND HMI Load All Defaults" %
%   N7:38  HT_PH_GAS_ALM_DLY  "CONFIG ADS Preheater Gas High Temp Alarm Delay" %
%   N7:39  HT_PH_GAS_WRN_DLY  "CONFIG ADS Preheater Gas High Temp Warning Delay" %
%   N7:40  HT_PH_GAS_ALM_SP  "CONFIG ADS Preheater Gas High Temp Alarm Setpoint" %
%   N7:41  HT_PH_GAS_WRN_SP  "CONFIG ADS Preheater Gas High Temp Warning Setpoint" %
%   N7:1/8  HT_PH_GAS_ALM_EN  "CONFIG ADS Preheater Gas High Temp Alarm Enable" %
%   N7:3/8  HT_PH_GAS_WRN_EN  "CONFIG ADS Preheater Gas High Temp Warning Enable" %

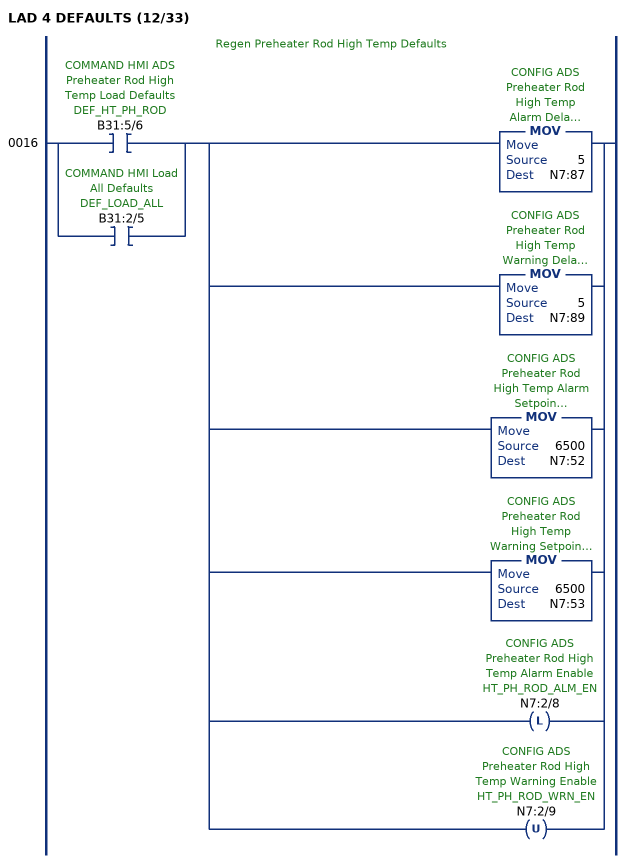
% Rung: 16 %
% Regen Preheater Rod High Temp Defaults %
SOR BST XIC B31:5/6 NXB XIC B31:2/5 BND BST MOV 5 N7:87 NXB MOV 5 N7:89 NXB MOV 6500 N7:52 NXB MOV 6500 N7:53 NXB OTL N7:2/8 NXB OTU N7:2/9 BND EOR
%   B31:5/6  DEF_HT_PH_ROD  "COMMAND HMI ADS Preheater Rod High Temp Load Defaults" %
%   B31:2/5  DEF_LOAD_ALL  "COMMAND HMI Load All Defaults" %
%   N7:87  HT_PH_ROD_ALM_DLY  "CONFIG ADS Preheater Rod High Temp Alarm Delay" %
%   N7:89  HT_PH_ROD_WRN_DLY  "CONFIG ADS Preheater Rod High Temp Warning Delay" %
%   N7:52  HT_PH_ROD_ALM_SP  "CONFIG ADS Preheater Rod High Temp Alarm Setpoint" %
%   N7:53  HT_PH_ROD_WRN_SP  "CONFIG ADS Preheater Rod High Temp Warning Setpoint" %
%   N7:2/8  HT_PH_ROD_ALM_EN  "CONFIG ADS Preheater Rod High Temp Alarm Enable" %
%   N7:2/9  HT_PH_ROD_WRN_EN  "CONFIG ADS Preheater Rod High Temp Warning Enable" %

